// TIA Portal project "项目1" (V14)

(* hardware
DEVICE "S7300/ET200M station_1"  S7-300 station
   slot 0: "导轨_0"  Rail  6ES7 390-1***0-0AA0
   slot 2: "PLC_1"  CPU 314C-2 PN/DP  6ES7 314-6EH04-0AB0  V3.3
      slot 2: "PROFINET 接口_1"  PN-IO
         slot 1: "Port_1"  Port
         slot 2: "Port_2"  Port
      slot 5: "DI 24/DO 16_1"  DI24/DO16
      slot 6: "AI 5/AO 2_1"  AI5/AO2
      slot 7: "计数_1"  Counter
      slot 8: "定位_1"  Positioning
*)

// ===== PLC "PLC_1"  CPU 314C-2 PN/DP =====

VAR_GLOBAL   // PLC tag table "变量表_1"
   "EW_L" AT %M0.4 : Bool;
   "EW_L_A" AT %Q4.6 : Bool;
   "EW_L_B" AT %Q4.7 : Bool;
   "EW_R_A" AT %Q5.2 : Bool;
   "EW_R_B" AT %Q5.3 : Bool;
   "EW_S" AT %M0.3 : Bool;
   "EW_S_A" AT %Q4.4 : Bool;
   "EW_S_B" AT %Q4.5 : Bool;
   "F_1Hz" AT %M10.5 : Bool;
   "SF" AT %M0.0 : Bool;
   "SN_L" AT %M0.2 : Bool;
   "SN_L_A" AT %Q4.2 : Bool;
   "SN_L_B" AT %Q4.3 : Bool;
   "SN_R_A" AT %Q5.0 : Bool;
   "SN_R_B" AT %Q5.1 : Bool;
   "SN_S" AT %M0.1 : Bool;
   "SN_S_A" AT %Q4.0 : Bool;
   "SN_S_B" AT %Q4.1 : Bool;
   "Start" AT %I0.0 : Bool;
   "Stop" AT %I0.1 : Bool;
   "T_0" AT %T0 : Timer;
   "T_1" AT %T1 : Timer;
   "T_10" AT %T10 : Timer;
   "T_11" AT %T11 : Timer;
   "T_12" AT %T12 : Timer;
   "T_13" AT %T13 : Timer;
   "T_14" AT %T14 : Timer;
   "T_15" AT %T15 : Timer;
   "T_2" AT %T2 : Timer;
   "T_3" AT %T3 : Timer;
   "T_4" AT %T4 : Timer;
   "T_5" AT %T5 : Timer;
   "T_6" AT %T6 : Timer;
   "T_7" AT %T7 : Timer;
   "T_8" AT %T8 : Timer;
   "T_9" AT %T9 : Timer;
END_VAR

TYPE "用户数据类型_1"
   STRUCT
      Element_1 : Int;
   END_STRUCT;
END_TYPE

DATA_BLOCK "FB1_DB"   // DB1
{ S7_Optimized_Access := 'FALSE' }
VERSION : 0.1
// stored: InstanceOfName FB1
"FB1"
BEGIN
END_DATA_BLOCK

DATA_BLOCK "FB1_DB_1"   // DB2
{ S7_Optimized_Access := 'FALSE' }
VERSION : 0.1
// stored: InstanceOfName FB1
"FB1"
BEGIN
END_DATA_BLOCK

DATA_BLOCK "FB1_DB_2"   // DB3
{ S7_Optimized_Access := 'FALSE' }
VERSION : 0.1
// stored: InstanceOfName FB1
"FB1"
BEGIN
END_DATA_BLOCK

DATA_BLOCK "FB1_DB_3"   // DB4
{ S7_Optimized_Access := 'FALSE' }
VERSION : 0.1
// stored: InstanceOfName FB1
"FB1"
BEGIN
END_DATA_BLOCK

FUNCTION_BLOCK "FB1"   // FB1, LAD
{ S7_Optimized_Access := 'FALSE' }
VERSION : 0.1
   VAR_INPUT
      R_ON : Bool;   // 控制变量，为0时亮红灯，为1时亮黄绿灯
      T_G : Timer;   // 绿灯常亮定时器
      T_Y : Timer;   // 黄灯常亮定时器
      T_GF : Timer;   // 绿灯闪烁定时器
      T_GW : S5Time;   // 绿灯常亮时间
      STOP : Bool;   // 停止信号
      F_1HZ : Bool;   // 1Hz时钟输入
   END_VAR
   VAR_OUTPUT
      LED_R : Bool;   // 亮红灯
      LED_G : Bool;   // 亮绿灯
      LED_Y : Bool;   // 亮黄灯
      "A" : Bool;   // 输出A
      "B" : Bool;   // 输出B
   END_VAR
   VAR
      T_GF_W : S5Time := S5T#3s;   // 绿灯闪烁时间
      T_Y_W : S5Time := S5T#2s;   // 黄灯常亮时间
   END_VAR
   VAR_TEMP
      tempr : Bool;
      tempy : Bool;
      tempg : Bool;
   END_VAR
   VAR_TEMP   // added for the SCL form of the ladder/FBD networks
      _w1 : Bool;
   END_VAR
BEGIN

REGION Network 1: 亮红灯
   // Network:1  当输入端R_ON状态为0时，应处于亮红灯的状态
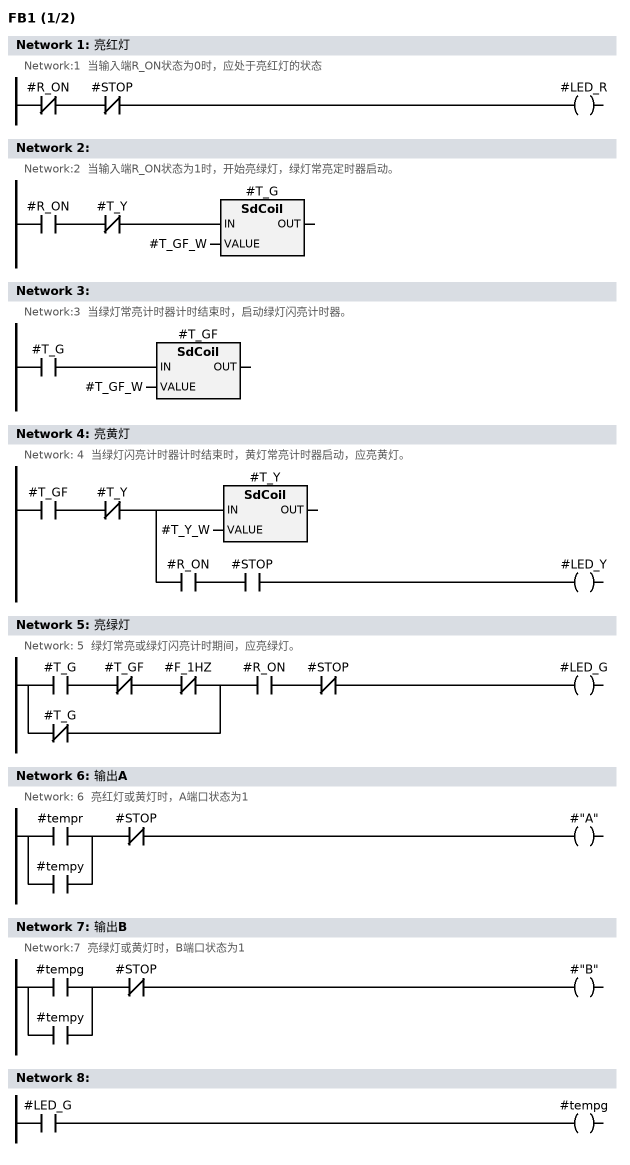
   RUNG wire#powerrail
      I_Contact( #R_ON )
      I_Contact( #STOP )
      Coil( #LED_R )
   END_RUNG
   // the same network as SCL:
   #LED_R := NOT #R_ON AND NOT #STOP;
END_REGION

REGION Network 2
   // Network:2  当输入端R_ON状态为1时，开始亮绿灯，绿灯常亮定时器启动。
   // no SCL statement known for SdCoil: written as a call
   SdCoil(in := #R_ON AND NOT #T_Y, value := #T_GF_W, operand := #T_G);
END_REGION

REGION Network 3
   // Network:3  当绿灯常亮计时器计时结束时，启动绿灯闪亮计时器。
   // no SCL statement known for SdCoil: written as a call
   SdCoil(in := #T_G, value := #T_GF_W, operand := #T_GF);
END_REGION

REGION Network 4: 亮黄灯
   // Network: 4  当绿灯闪亮计时器计时结束时，黄灯常亮计时器启动，应亮黄灯。
   // no SCL statement known for SdCoil: written as a call
   #_w1 := #T_GF AND NOT #T_Y;
   SdCoil(in := #_w1, value := #T_Y_W, operand := #T_Y);
   #LED_Y := #_w1 AND #R_ON AND #STOP;
END_REGION

REGION Network 5: 亮绿灯
   // Network: 5  绿灯常亮或绿灯闪亮计时期间，应亮绿灯。
   RUNG wire#powerrail
      Contact( #T_G )
      I_Contact( #T_GF )
      I_Contact( #F_1HZ )
      wire#w1
      Contact( #R_ON )
      I_Contact( #STOP )
      Coil( #LED_G )
   END_RUNG
   RUNG wire#powerrail
      I_Contact( #T_G )
   END_RUNG wire#w1
   // the same network as SCL:
   #LED_G := ((#T_G AND NOT #T_GF AND NOT #F_1HZ) OR NOT #T_G) AND #R_ON AND NOT #STOP;
END_REGION

REGION Network 6: 输出A
   // Network: 6  亮红灯或黄灯时，A端口状态为1
   RUNG wire#powerrail
      Contact( #tempr )
      wire#w1
      I_Contact( #STOP )
      Coil( #"A" )
   END_RUNG
   RUNG wire#powerrail
      Contact( #tempy )
   END_RUNG wire#w1
   // the same network as SCL:
   #"A" := (#tempr OR #tempy) AND NOT #STOP;
END_REGION

REGION Network 7: 输出B
   // Network:7  亮绿灯或黄灯时，B端口状态为1
   RUNG wire#powerrail
      Contact( #tempg )
      wire#w1
      I_Contact( #STOP )
      Coil( #"B" )
   END_RUNG
   RUNG wire#powerrail
      Contact( #tempy )
   END_RUNG wire#w1
   // the same network as SCL:
   #"B" := (#tempg OR #tempy) AND NOT #STOP;
END_REGION

REGION Network 8
   RUNG wire#powerrail
      Contact( #LED_G )
      Coil( #tempg )
   END_RUNG
   // the same network as SCL:
   #tempg := #LED_G;
END_REGION

REGION Network 9
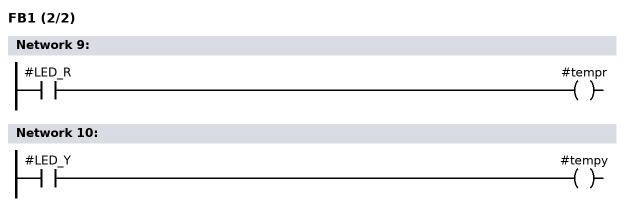
   RUNG wire#powerrail
      Contact( #LED_R )
      Coil( #tempr )
   END_RUNG
   // the same network as SCL:
   #tempr := #LED_R;
END_REGION

REGION Network 10
   RUNG wire#powerrail
      Contact( #LED_Y )
      Coil( #tempy )
   END_RUNG
   // the same network as SCL:
   #tempy := #LED_Y;
END_REGION
END_FUNCTION_BLOCK

ORGANIZATION_BLOCK "Main"   // OB1, LAD
TITLE = "Main Program Sweep (Cycle)"
{ S7_Optimized_Access := 'FALSE' }
VERSION : 0.1
   VAR_TEMP
      OB1_EV_CLASS : Byte;   // Bits 0-3 = 1 (Coming event), Bits 4-7 = 1 (Event class 1)
      OB1_SCAN_1 : Byte;   // 1 (Cold restart scan 1 of OB 1), 3 (Scan 2-n of OB 1)
      OB1_PRIORITY : Byte;   // Priority of OB Execution
      OB1_OB_NUMBR : Byte;   // 1 (Organization block 1, OB1)
      OB1_RESERVED_1 : Byte;   // Reserved for system
      OB1_RESERVED_2 : Byte;   // Reserved for system
      OB1_PREV_CYCLE : Int;   // Cycle time of previous OB1 scan (milliseconds)
      OB1_MIN_CYCLE : Int;   // Minimum cycle time of OB1 (milliseconds)
      OB1_MAX_CYCLE : Int;   // Maximum cycle time of OB1 (milliseconds)
      OB1_DATE_TIME : Date_And_Time;   // Date and time OB1 started
   END_VAR
   VAR_TEMP   // added for the SCL form of the ladder/FBD networks
      _w1 : Bool;
   END_VAR
BEGIN

REGION Network 1: 常开按钮
   // Network:1 根据启动按钮和停止按钮确定启动状态SF
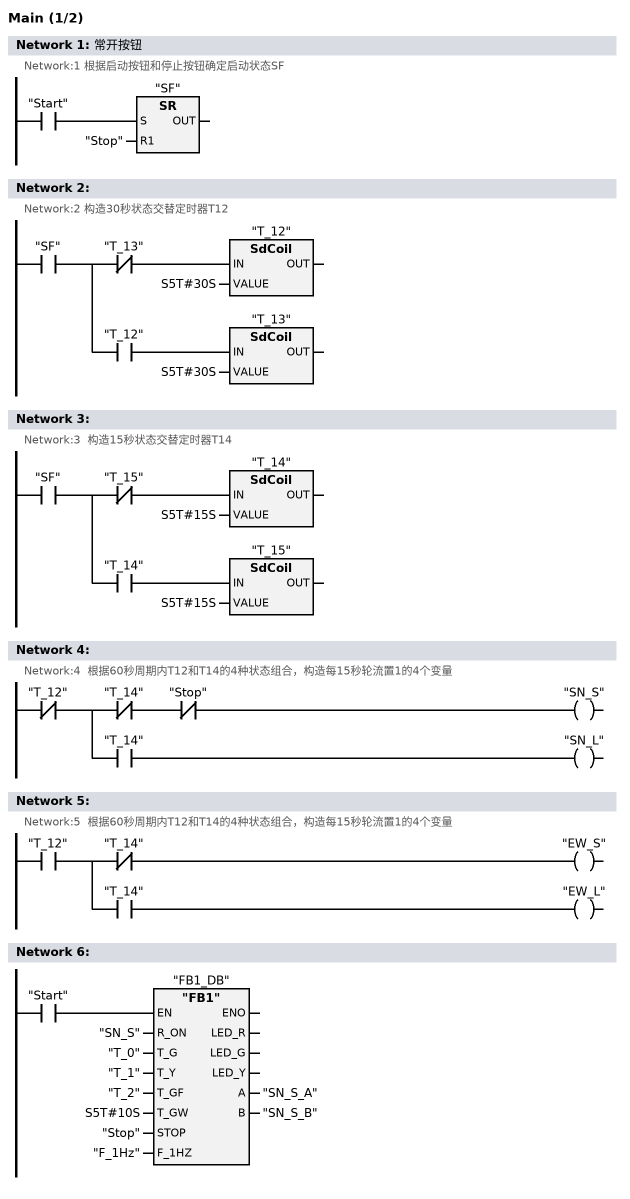
   RUNG wire#powerrail
      Contact( "Start" )
      S_SR(operand := "SF", r1 := "Stop")
   END_RUNG
   // the same network as SCL:
   IF "Start" THEN
       "SF" := TRUE;   // SR flip-flop
   END_IF;
   IF "Stop" THEN "SF" := FALSE; END_IF;
END_REGION

REGION Network 2
   // Network:2 构造30秒状态交替定时器T12
   // no SCL statement known for SdCoil: written as a call
   #_w1 := "SF";
   SdCoil(in := "SF" AND NOT "T_13", value := S5T#30S, operand := "T_12");
   SdCoil(in := #_w1 AND "T_12", value := S5T#30S, operand := "T_13");
END_REGION

REGION Network 3
   // Network:3  构造15秒状态交替定时器T14
   // no SCL statement known for SdCoil: written as a call
   #_w1 := "SF";
   SdCoil(in := "SF" AND NOT "T_15", value := S5T#15S, operand := "T_14");
   SdCoil(in := #_w1 AND "T_14", value := S5T#15S, operand := "T_15");
END_REGION

REGION Network 4
   // Network:4  根据60秒周期内T12和T14的4种状态组合，构造每15秒轮流置1的4个变量
   RUNG wire#powerrail
      I_Contact( "T_12" )
      wire#w1
      I_Contact( "T_14" )
      I_Contact( "Stop" )
      Coil( "SN_S" )
   END_RUNG
   RUNG wire#w1
      Contact( "T_14" )
      Coil( "SN_L" )
   END_RUNG
   // the same network as SCL:
   "SN_S" := NOT "T_12" AND NOT "T_14" AND NOT "Stop";
   "SN_L" := NOT "T_12" AND "T_14";
END_REGION

REGION Network 5
   // Network:5  根据60秒周期内T12和T14的4种状态组合，构造每15秒轮流置1的4个变量
   RUNG wire#powerrail
      Contact( "T_12" )
      wire#w1
      I_Contact( "T_14" )
      Coil( "EW_S" )
   END_RUNG
   RUNG wire#w1
      Contact( "T_14" )
      Coil( "EW_L" )
   END_RUNG
   // the same network as SCL:
   "EW_S" := "T_12" AND NOT "T_14";
   "EW_L" := "T_12" AND "T_14";
END_REGION

REGION Network 6
   RUNG wire#powerrail
      Contact( "Start" )
      "FB1_DB"(R_ON := "SN_S", T_G := "T_0", T_Y := "T_1", T_GF := "T_2", T_GW := S5T#10S, STOP := "Stop", F_1HZ := "F_1Hz", LED_R =>, LED_G =>, LED_Y =>, "A" => "SN_S_A", "B" => "SN_S_B")
   END_RUNG
   // the same network as SCL:
   IF "Start" THEN
       "FB1_DB"(R_ON := "SN_S",   // "FB1"
                T_G := "T_0",
                T_Y := "T_1",
                T_GF := "T_2",
                T_GW := S5T#10S,
                STOP := "Stop",
                F_1HZ := "F_1Hz",
                "A" => "SN_S_A",
                "B" => "SN_S_B");
   END_IF;
END_REGION

REGION Network 7
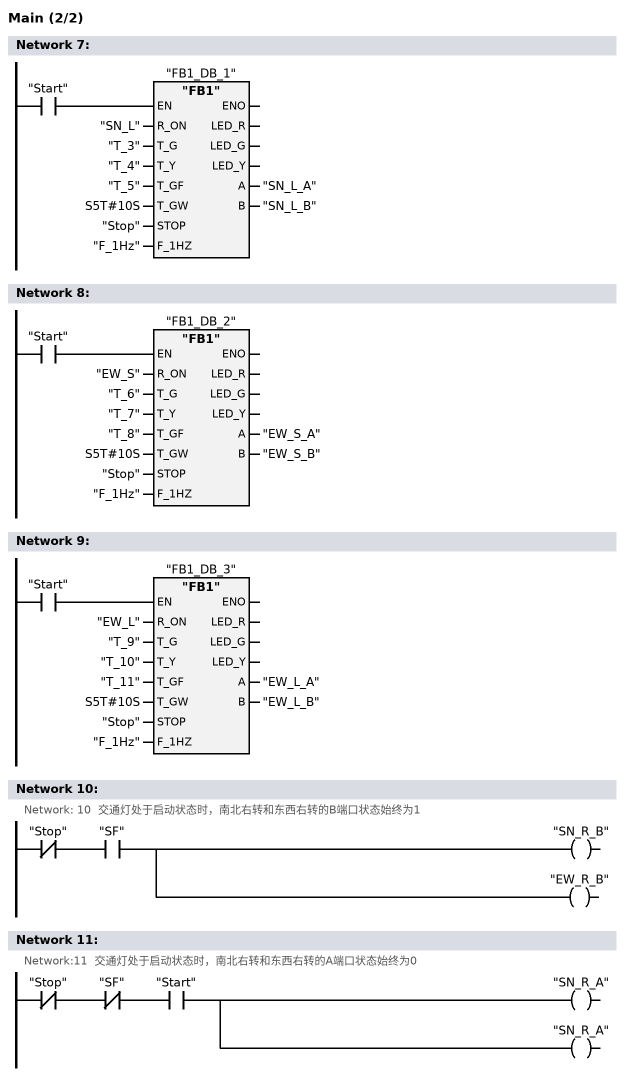
   RUNG wire#powerrail
      Contact( "Start" )
      "FB1_DB_1"(R_ON := "SN_L", T_G := "T_3", T_Y := "T_4", T_GF := "T_5", T_GW := S5T#10S, STOP := "Stop", F_1HZ := "F_1Hz", LED_R =>, LED_G =>, LED_Y =>, "A" => "SN_L_A", "B" => "SN_L_B")
   END_RUNG
   // the same network as SCL:
   IF "Start" THEN
       "FB1_DB_1"(R_ON := "SN_L",   // "FB1"
                  T_G := "T_3",
                  T_Y := "T_4",
                  T_GF := "T_5",
                  T_GW := S5T#10S,
                  STOP := "Stop",
                  F_1HZ := "F_1Hz",
                  "A" => "SN_L_A",
                  "B" => "SN_L_B");
   END_IF;
END_REGION

REGION Network 8
   RUNG wire#powerrail
      Contact( "Start" )
      "FB1_DB_2"(R_ON := "EW_S", T_G := "T_6", T_Y := "T_7", T_GF := "T_8", T_GW := S5T#10S, STOP := "Stop", F_1HZ := "F_1Hz", LED_R =>, LED_G =>, LED_Y =>, "A" => "EW_S_A", "B" => "EW_S_B")
   END_RUNG
   // the same network as SCL:
   IF "Start" THEN
       "FB1_DB_2"(R_ON := "EW_S",   // "FB1"
                  T_G := "T_6",
                  T_Y := "T_7",
                  T_GF := "T_8",
                  T_GW := S5T#10S,
                  STOP := "Stop",
                  F_1HZ := "F_1Hz",
                  "A" => "EW_S_A",
                  "B" => "EW_S_B");
   END_IF;
END_REGION

REGION Network 9
   RUNG wire#powerrail
      Contact( "Start" )
      "FB1_DB_3"(R_ON := "EW_L", T_G := "T_9", T_Y := "T_10", T_GF := "T_11", T_GW := S5T#10S, STOP := "Stop", F_1HZ := "F_1Hz", LED_R =>, LED_G =>, LED_Y =>, "A" => "EW_L_A", "B" => "EW_L_B")
   END_RUNG
   // the same network as SCL:
   IF "Start" THEN
       "FB1_DB_3"(R_ON := "EW_L",   // "FB1"
                  T_G := "T_9",
                  T_Y := "T_10",
                  T_GF := "T_11",
                  T_GW := S5T#10S,
                  STOP := "Stop",
                  F_1HZ := "F_1Hz",
                  "A" => "EW_L_A",
                  "B" => "EW_L_B");
   END_IF;
END_REGION

REGION Network 10
   // Network: 10  交通灯处于启动状态时，南北右转和东西右转的B端口状态始终为1
   RUNG wire#powerrail
      I_Contact( "Stop" )
      Contact( "SF" )
      wire#w1
      Coil( "SN_R_B" )
   END_RUNG
   RUNG wire#w1
      Coil( "EW_R_B" )
   END_RUNG
   // the same network as SCL:
   "SN_R_B" := NOT "Stop" AND "SF";
   "EW_R_B" := "SN_R_B";
END_REGION

REGION Network 11
   // Network:11  交通灯处于启动状态时，南北右转和东西右转的A端口状态始终为0
   RUNG wire#powerrail
      I_Contact( "Stop" )
      I_Contact( "SF" )
      Contact( "Start" )
      wire#w1
      Coil( "SN_R_A" )
   END_RUNG
   RUNG wire#w1
      Coil( "SN_R_A" )
   END_RUNG
   // the same network as SCL:
   "SN_R_A" := NOT "Stop" AND NOT "SF" AND "Start";
   "SN_R_A" := "SN_R_A";
END_REGION
END_ORGANIZATION_BLOCK

ORGANIZATION_BLOCK "COMPLETE RESTART"   // OB100, LAD
TITLE = "Complete Restart"
{ S7_Optimized_Access := 'FALSE' }
VERSION : 0.1
   VAR_TEMP
      OB100_EV_CLASS : Byte;   // 16#13, Event class 1, Entering event state, Event logged in diagnostic buffer
      OB100_STRTUP : Byte;   // 16#81/82/83/84 Method of startup
      OB100_PRIORITY : Byte;   // Priority of OB Execution
      OB100_OB_NUMBR : Byte;   // 100 (Organization block 100, OB100)
      OB100_RESERVED_1 : Byte;   // Reserved for system
      OB100_RESERVED_2 : Byte;   // Reserved for system
      OB100_STOP : Word;   // Event that caused CPU to stop (16#4xxx)
      OB100_STRT_INFO : DWord;   // Information on how system started
      OB100_DATE_TIME : Date_And_Time;   // Date and time OB100 started
   END_VAR
BEGIN

REGION Network 1
   // Network:1  启动按钮未打卡前，所有输出状态置0
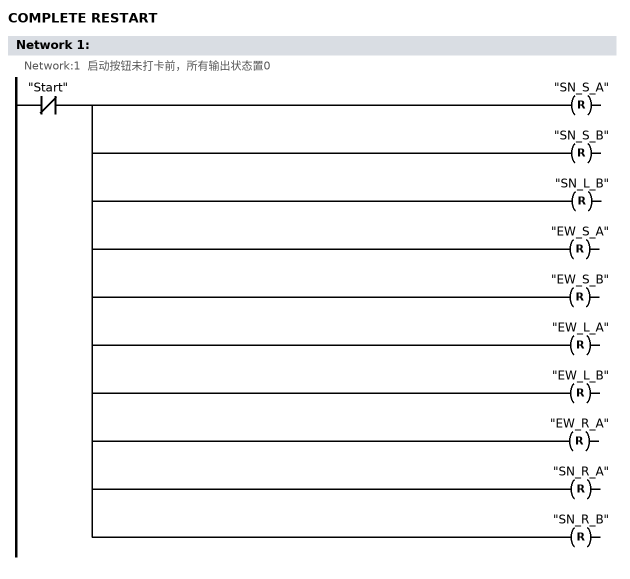
   RUNG wire#powerrail
      I_Contact( "Start" )
      wire#w1
      R_Coil( "SN_S_A" )
   END_RUNG
   RUNG wire#w1
      R_Coil( "SN_S_B" )
   END_RUNG
   RUNG wire#w1
      R_Coil( "SN_L_B" )
   END_RUNG
   RUNG wire#w1
      R_Coil( "EW_S_A" )
   END_RUNG
   RUNG wire#w1
      R_Coil( "EW_S_B" )
   END_RUNG
   RUNG wire#w1
      R_Coil( "EW_L_A" )
   END_RUNG
   RUNG wire#w1
      R_Coil( "EW_L_B" )
   END_RUNG
   RUNG wire#w1
      R_Coil( "EW_R_A" )
   END_RUNG
   RUNG wire#w1
      R_Coil( "SN_R_A" )
   END_RUNG
   RUNG wire#w1
      R_Coil( "SN_R_B" )
   END_RUNG
   // the same network as SCL:
   IF NOT "Start" THEN
       "SN_S_A" := FALSE;
       "SN_S_B" := FALSE;
       "SN_L_B" := FALSE;
       "EW_S_A" := FALSE;
       "EW_S_B" := FALSE;
       "EW_L_A" := FALSE;
       "EW_L_B" := FALSE;
       "EW_R_A" := FALSE;
       "SN_R_A" := FALSE;
       "SN_R_B" := FALSE;
   END_IF;
END_REGION
END_ORGANIZATION_BLOCK